# B&R Automation Studio project VerticalStacker
Automation Studio 4.10.2.37; technology packages: mappMotion 5.12.3, mappSafety 5.12.2

## Configuration Simulation

CPU X20cCP3586, AutomationRuntime B4.91, Build 4.1.2, Safety 0.0, Vc V4.72.3

### Task classes (Cpu.sw)
```
Cyclic#1:
  Program <- Program.prg
Libraries: SfDomain, standard, McBase, MpAxis, McAxis, MpBase, McAcpAx
```

### Hardware
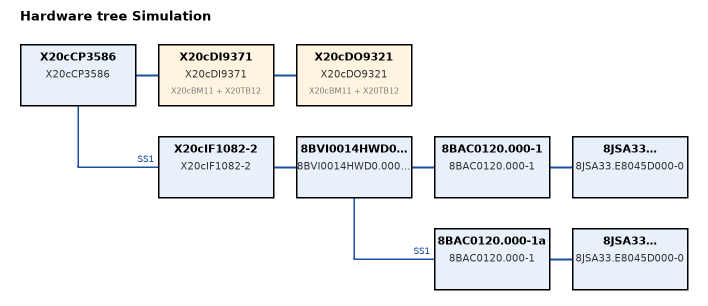
```
8BAC0120.000-1 : 8BAC0120.000-1 v2.2.0.0  [SS -> 8BVI0014HWD0.000-1.SS2]
  PlugInType = Encoder
  McAcoposTypeID = AcoposMultiPlugInConfig
8BAC0120.000-1a : 8BAC0120.000-1 v2.2.0.0  [SS -> 8BVI0014HWD0.000-1.SS1]
  PlugInType = Encoder
  McAcoposTypeID = AcoposMultiPlugInConfig
8BVI0014HWD0.000-1 : 8BVI0014HWD0.000-1 v2.3.0.1  [PLK1 -> X20cIF1082-2.IF1 (NodeNumber=1) [Cable Type=PowerlinkCable, Length=10, Version=1.0.0.3]; MT2 -> 8JSA33.E8045D000-0.MT]
  DriveConfiguration/Module:
    McAcoposTypeID = AcoposMultiDConfig
    ActivateACOPOSSimulationOnPLC = 1
    PowerSupply = ETA
  DriveConfiguration/Channel[1]/RealAxis:
    AxisReference = 
  DriveConfiguration/Channel[1]/RealAxis/MechanicalElements/Gearbox:
    InputIsReadOnly = 0
    Input = 1
    OutputIsReadOnly = 0
    Output = 1
  DriveConfiguration/Channel[1]/RealAxis/MechanicalElements/RotaryToLinearTransformation:
    ReferenceDistanceIsReadOnly = 0
    ReferenceDistance = 1
  DriveConfiguration/Channel[1]/RealAxis/Controller:
    ModeIsReadOnly = 0
    Mode = PositionController
  DriveConfiguration/Channel[1]/RealAxis/Controller/Mode/Position:
    ProportionalGain = 50.0
    IntegrationTime = 0.0
    PredictionTime = 0.0004
    TotalDelayTime = 0.0004
  DriveConfiguration/Channel[1]/RealAxis/Controller/Mode/Speed:
    ProportionalGainIsReadOnly = 0
    ProportionalGain = 2.0
    IntegrationTimeIsReadOnly = 0
    IntegrationTime = 0.0
    FilterTimeIsReadOnly = 0
    FilterTime = 0.0
  DriveConfiguration/Channel[1]/RealAxis/Controller/Mode/LoopFilters:
    LoopFilter1 = NotUsed
    LoopFilter2 = NotUsed
    LoopFilter3 = NotUsed
  DriveConfiguration/Channel[1]/RealAxis/Homing:
    Mode = Direct
  DriveConfiguration/Channel[1]/RealAxis/Homing/Mode:
    Position = 0.0
    ReferencePulse = NotUsed
  DriveConfiguration/Channel[1]/RealAxis/Homing:
    RestorePositionVariable = 
  DriveConfiguration/Channel[1]/RealAxis/StopReaction:
    Quickstop = DecelerationLimit
    DriveError = DecelerationLimit
  DriveConfiguration/Channel[1]/RealAxis/MovementErrorLimits:
    PositionError = 1.0
    VelocityErrorMonitoring = Automatic1
  DriveConfiguration/Channel[1]/RealAxis:
    JerkFilter = NotUsed
  DriveConfiguration/Channel[1]/RealAxis/DigitalInputs/HomingSwitch:
    Source = NotUsed
    Level = High
  DriveConfiguration/Channel[1]/RealAxis/DigitalInputs/PositiveLimitSwitch:
    Source = NotUsed
    Level = High
  DriveConfiguration/Channel[1]/RealAxis/DigitalInputs/NegativeLimitSwitch:
    Source = NotUsed
    Level = High
  DriveConfiguration/Channel[1]/RealAxis/DigitalInputs/Trigger1:
    Level = High
  DriveConfiguration/Channel[1]/RealAxis/DigitalInputs/Trigger2:
    Level = High
  DriveConfiguration/Channel[1]/RealAxis/DigitalInputs/Quickstop:
    Input = Trigger2
  DriveConfiguration/Channel[1]/RealAxis/Simulation:
    SimulationModeOnPLC = SetValueGeneration
    SimulationModeOnACOPOS = NotUsed
  DriveConfiguration/Channel[1]:
    VirtualAxis = Used
  DriveConfiguration/Channel[1]/VirtualAxis:
    AxisReference = gAxis_1
  DriveConfiguration/Channel[1]/VirtualAxis/Homing:
    Mode = Direct
  DriveConfiguration/Channel[1]/VirtualAxis/Homing/Mode:
    Position = 0.0
  DriveConfiguration/Channel[1]/VirtualAxis/Homing:
    RestorePositionVariable = 
  DriveConfiguration/Channel[1]/VirtualAxis:
    JerkFilter = NotUsed
  DriveConfiguration/Channel[2]/RealAxis:
    AxisReference = 
  DriveConfiguration/Channel[2]/RealAxis/MechanicalElements/Gearbox:
    InputIsReadOnly = 0
    Input = 1
    OutputIsReadOnly = 0
    Output = 1
  DriveConfiguration/Channel[2]/RealAxis/MechanicalElements/RotaryToLinearTransformation:
    ReferenceDistanceIsReadOnly = 0
    ReferenceDistance = 1
  DriveConfiguration/Channel[2]/RealAxis/Controller:
    ModeIsReadOnly = 0
    Mode = PositionController
  DriveConfiguration/Channel[2]/RealAxis/Controller/Mode/Position:
    ProportionalGain = 50.0
    IntegrationTime = 0.0
    PredictionTime = 0.0004
    TotalDelayTime = 0.0004
  DriveConfiguration/Channel[2]/RealAxis/Controller/Mode/Speed:
    ProportionalGainIsReadOnly = 0
    ProportionalGain = 2.0
    IntegrationTimeIsReadOnly = 0
    IntegrationTime = 0.0
    FilterTimeIsReadOnly = 0
    FilterTime = 0.0
  DriveConfiguration/Channel[2]/RealAxis/Controller/Mode/LoopFilters:
    LoopFilter1 = NotUsed
    LoopFilter2 = NotUsed
    LoopFilter3 = NotUsed
  DriveConfiguration/Channel[2]/RealAxis/Homing:
    Mode = Direct
  DriveConfiguration/Channel[2]/RealAxis/Homing/Mode:
    Position = 0.0
    ReferencePulse = NotUsed
  DriveConfiguration/Channel[2]/RealAxis/Homing:
    RestorePositionVariable = 
  DriveConfiguration/Channel[2]/RealAxis/StopReaction:
    Quickstop = DecelerationLimit
    DriveError = DecelerationLimit
  DriveConfiguration/Channel[2]/RealAxis/MovementErrorLimits:
    PositionError = 1.0
    VelocityErrorMonitoring = Automatic1
  DriveConfiguration/Channel[2]/RealAxis:
    JerkFilter = NotUsed
  DriveConfiguration/Channel[2]/RealAxis/DigitalInputs/HomingSwitch:
    Source = NotUsed
    Level = High
  DriveConfiguration/Channel[2]/RealAxis/DigitalInputs/PositiveLimitSwitch:
    Source = NotUsed
    Level = High
  DriveConfiguration/Channel[2]/RealAxis/DigitalInputs/NegativeLimitSwitch:
    Source = NotUsed
    Level = High
  DriveConfiguration/Channel[2]/RealAxis/DigitalInputs/Trigger1:
    Level = High
  DriveConfiguration/Channel[2]/RealAxis/DigitalInputs/Trigger2:
    Level = High
  DriveConfiguration/Channel[2]/RealAxis/DigitalInputs/Quickstop:
    Input = Trigger2
  DriveConfiguration/Channel[2]/RealAxis/Simulation:
    SimulationModeOnPLC = SetValueGeneration
    SimulationModeOnACOPOS = NotUsed
  DriveConfiguration/Channel[2]:
    VirtualAxis = Used
  DriveConfiguration/Channel[2]/VirtualAxis:
    AxisReference = gAxis_2
  DriveConfiguration/Channel[2]/VirtualAxis/Homing:
    Mode = Direct
  DriveConfiguration/Channel[2]/VirtualAxis/Homing/Mode:
    Position = 0.0
  DriveConfiguration/Channel[2]/VirtualAxis/Homing:
    RestorePositionVariable = 
  DriveConfiguration/Channel[2]/VirtualAxis:
    JerkFilter = NotUsed
8JSA33.E8045D000-0 : 8JSA33.E8045D000-0 v1.0.6.30  [EC -> 8BAC0120.000-1.EC; MT -> 8BVI0014HWD0.000-1.MT2]
8JSA33.E8045D000-0a : 8JSA33.E8045D000-0 v1.0.6.30  [EC -> 8BAC0120.000-1a.EC; MT -> 8BVI0014HWD0.000-1.MT1]
X20TB12 : X20TB12 v1.0.0.0
X20TB12a : X20TB12 v1.0.0.0
X20cBM11 : X20cBM11 v1.0.1.0  [X2X1 -> X20cCP3586.IF6]
X20cBM11a : X20cBM11 v1.0.1.0  [X2X1 -> X20cBM11.X2X2]
X20cCP3586 : X20cCP3586 v1.9.0.0
  Connector IF2:
    ActivateDevice = 1
  ConfigurationID = Project_VerticalStacker_Config1
  Simulation = 1
  FileDevice1
  FileDeviceName1 = USER
  FileDevicePath1 = USER_PATH
  ActivateOpcUa = 1
  OpcUaPort = 4842
  OpcUa_AuthenticationSecurityPolicy_EnableNone = 1
  OpcUa_AuthenticationSecurityPolicy_EnableBasic128Rsa15 = 1
  OpcUaInformationModels_PV_Version = 1
X20cDI9371 : X20cDI9371 v1.1.0.0  [SS1 -> X20TB12.SS; SL -> X20cBM11.SL1]
X20cDO9321 : X20cDO9321 v1.1.0.0  [SS1 -> X20TB12a.SS; SL -> X20cBM11a.SL1]
X20cIF1082-2 : X20cIF1082-2 v1.11.1.0  [SS -> X20cCP3586.SS1]
  Connector IF1:
    EplNatSubnet = 192.168.102.0
```

- Physical/Simulation/X20cCP3586/IoMap.iom: same as Physical/Simulation/X20cCP3586/Cpu.per
- Physical/Simulation/X20cCP3586/PvMap.vvm: same as Physical/Simulation/X20cCP3586/Cpu.per
### Config_1.axis - X20cCP3586/mappMotion/Config_1.axis
```
Element gAxis_1 (Type=axis)
  BaseTypeIsReadOnly = 0
  BaseType = LinearBounded
    MeasurementUnit = 5066068
    MeasurementResolutionIsReadOnly = 0
    MeasurementResolution = 0.01
    CountDirectionIsReadOnly = 0
    CountDirection = Standard
  MovementLimitsIsReadOnly = 0
  MovementLimits = Internal
    Position:
      LowerLimitMin = -1.79769313486231E308
      UpperLimitMax = 1.79769313486231E308
      LowerLimit = -1000.0
      UpperLimit = 1000.0
    VelocityIsReadOnly = 0
    Velocity:
      VelocityMax = 3.4E38
      Velocity = 10.0
    AccelerationIsReadOnly = 0
    Acceleration:
      AccelerationMax = 3.4E38
      Acceleration = 50.0
    DecelerationIsReadOnly = 0
    Deceleration:
      DecelerationMax = 3.4E38
      Deceleration = 50.0
  Alarms = None
Element gAxis_2 (Type=axis)
  BaseTypeIsReadOnly = 0
  BaseType = LinearBounded
    MeasurementUnit = 5066068
    MeasurementResolutionIsReadOnly = 0
    MeasurementResolution = 0.01
    CountDirectionIsReadOnly = 0
    CountDirection = Standard
  MovementLimitsIsReadOnly = 0
  MovementLimits = Internal
    Position:
      LowerLimitMin = -1.79769313486231E308
      UpperLimitMax = 1.79769313486231E308
      LowerLimit = -1000.0
      UpperLimit = 1000.0
    VelocityIsReadOnly = 0
    Velocity:
      VelocityMax = 3.4E38
      Velocity = 10.0
    AccelerationIsReadOnly = 0
    Acceleration:
      AccelerationMax = 3.4E38
      Acceleration = 50.0
    DecelerationIsReadOnly = 0
    Deceleration:
      DecelerationMax = 3.4E38
      Deceleration = 50.0
  Alarms = None
```

- Safety project (password-protected, skipped)

## Logical view

Binary libraries used (declarations not repeated): operator, runtime, astime, AsIecCon, SfDomain 5.12.2, standard, McBase 5.12.3, MpAxis 5.12.3, McAxis 5.12.3, MpBase 5.12.0, McAcpAx 5.12.3


### Program Logical/Program (IEC)

#### Main.st - Init, cyclic, exit code
```iecst
(*
Name					Date				Version				Note
Jamal Muhammad			10.10.2021			V2021.1				First version
*)

PROGRAM _INIT
	MpAxisBasic_0.Enable := TRUE;
	xHomingCmd := TRUE;

	AxisParameters.Velocity := 5.0;
	AxisParameters.Acceleration := 20.0;
	AxisParameters.Deceleration := 20.0;

	xPartLoadFirstCycle := TRUE;
	xPartUnloadFirstCycle := TRUE;
	// For simulation purpose
	FOR i:=1 TO 20 DO
		aBufferData[i].usiSeqNumber:= i;
		aBufferData[i].usiPartId := 100+i;
	END_FOR
	usiPartId := 120;
END_PROGRAM

PROGRAM _CYCLIC
	// Inputs
	lrServoPosition := MpAxisBasic_0.Position;

	stServoState.PowerON := MpAxisBasic_0.PowerOn;
	stServoState.Active := MpAxisBasic_0.Active;
	stServoState.MoveActive := MpAxisBasic_0.MoveActive;
	stServoState.Error := MpAxisBasic_0.Error;

	// Initialisation
	IF xInit = FALSE THEN
		ton_1(IN:=NOT ton_1.Q,PT:=T#3500MS);
		IF ton_1.Q THEN
			ton_1(IN:=FALSE,PT:=t#0MS);
			xInit := TRUE;
		END_IF
	END_IF

	//	Enabling/Disabling servo
	IF xServoError OR xEmergencyStopInactive_NC=FALSE OR xDriveStopInactive_NC=FALSE THEN
		xServoEnable:=FALSE;
	ELSE
		xServoEnable:=TRUE;
	END_IF

	// Enabling servo power automatically after initialisation & xServoEnable are ON
	IF xServoEnable AND xInit AND MpAxisBasic_0.PowerOn = FALSE THEN
		MpAxisBasic_0.Power := TRUE;
	END_IF

	// If xHomingCmd is ON then move servo to zero position
	IF MpAxisBasic_0.Position = 0 THEN
		xHomingCmd := FALSE;
	ELSIF MpAxisBasic_0.Position<>0 AND xHomingCmd = TRUE AND MpAxisBasic_0.PowerOn THEN
		AxisParameters.Position := 0.0;
		MpAxisBasic_0.MoveAbsolute := TRUE;
	END_IF;

	// Part unloading has priority-1, part unloading has priority-2
	IF xUnloadPartCmd THEN
		xLoadPartCmd := FALSE;
	END_IF

	//Check if buffer is full
	usiCounter := 0;
	FOR i:=1 TO usiPartBufferMax DO
		IF aBufferData[i].usiPartId <> 0 THEN
			usiCounter := usiCounter+1;
		END_IF
	END_FOR
	IF usiCounter = usiPartBufferMax THEN
		xBufferFull:=TRUE;
	ELSE
		xBufferFull:=FALSE;
	END_IF

	// State Machine > Unloading buffer
	IF xUnloadPartCmd AND xHomingCmd=FALSE AND MpAxisBasic_0.Enable THEN
		enumState_part_loading:=ST_LD_TO_ZERO_POS_1;
		xPartLoadFirstCycle:=TRUE;

		CASE enumState_part_unloading OF
			//*********************
			ST_UNLD_TO_ZERO_POS_1:
				IF xPartUnloadFirstCycle AND lrServoPosition<>0 THEN
					AxisParameters.Position := 0.0;
					AxisParameters.Velocity := 40.0;
					AxisParameters.Acceleration := 160.0;
					AxisParameters.Deceleration := 160.0;
					AxisUpdate;
					IF xAxisUpdateDone AND MpAxisBasic_0.MoveActive=FALSE THEN
						MpAxisBasic_0.MoveAbsolute := TRUE;
						enumState_part_unloading:=ST_UNLD_TO_ZERO_POS_2;
					END_IF
				ELSE
					enumState_part_unloading:=ST_UNLD_SET_AXIS_PARAMS_1;
				END_IF
			//*********************
			ST_UNLD_TO_ZERO_POS_2:
				IF lrServoPosition=0 THEN
					xPartUnloadFirstCycle := FALSE;
					MpAxisBasic_0.MoveAbsolute := FALSE;
					enumState_part_unloading:=ST_UNLD_SET_AXIS_PARAMS_1;
				END_IF
			//*********************
			ST_UNLD_SET_AXIS_PARAMS_1:
				IF lrServoPosition<690 AND MpAxisBasic_0.MoveActive=FALSE THEN
					AxisParameters.Position := 690.0;
					AxisParameters.Velocity := 10.0;
					AxisParameters.Acceleration := 40.0;
					AxisParameters.Deceleration := 40.0;
					AxisUpdate;
					IF xAxisUpdateDone THEN
						enumState_part_unloading:=ST_UNLD_IF_UNLOAD_CMD;
					END_IF
				END_IF
			//*********************
			ST_UNLD_IF_UNLOAD_CMD:
				IF xUnloadPartCmd THEN
					enumState_part_unloading:=ST_UNLD_FIND_UNLOADING_TARGET;
				END_IF
			//*********************
			ST_UNLD_FIND_UNLOADING_TARGET:
				FOR i:=1 TO usiPartBufferMax DO
					IF aBufferData[i].usiPartId <> 0 THEN
						FOR j:=1 TO usiPartBufferMax DO
							IF aBufferData[j].usiPartId<>0 AND i<>j AND aBufferData[i].usiPartId < aBufferData[j].usiPartId THEN
								usiTarget := i;
							ELSIF i=usiPartBufferMax THEN
								usiTarget := i;
							ELSE
								usiTarget := 0;
							END_IF
						END_FOR
						IF usiTarget<>0 THEN
							enumState_part_unloading:=ST_UNLD_SET_AXIS_PARAMS_2;
							EXIT;
						END_IF
					END_IF
				END_FOR
			//*********************
			ST_UNLD_SET_AXIS_PARAMS_2:
				AxisParameters.Position := usiTarget*34.5;
				AxisParameters.Velocity := 10.0;
				AxisParameters.Acceleration := 40.0;
				AxisParameters.Deceleration := 40.0;
				IF xAxisUpdateDone THEN
					enumState_part_unloading:=ST_UNLD_SERVO_MOVE_TO_TARGET;
				END_IF
			//*********************
			ST_UNLD_SERVO_MOVE_TO_TARGET:
				MpAxisBasic_0.MoveAbsolute := TRUE;

				IF AxisParameters.Position > lrServoPosition  THEN
					IF lrServoPosition > AxisParameters.Position-5 THEN
						MpAxisBasic_0.MoveAbsolute := FALSE;
						enumState_part_unloading:=ST_UNLD_SET_AXIS_PARAMS_3;
					END_IF;
				END_IF

				IF AxisParameters.Position < lrServoPosition  THEN
					IF lrServoPosition < AxisParameters.Position+5 THEN
						MpAxisBasic_0.MoveAbsolute := FALSE;
						enumState_part_unloading:=ST_UNLD_SET_AXIS_PARAMS_3;
					END_IF;
				END_IF
			//*********************
			ST_UNLD_SET_AXIS_PARAMS_3:
				IF MpAxisBasic_0.MoveActive = FALSE THEN
					AxisParameters.Velocity := 1.0;
					AxisParameters.Acceleration := 4.0;
					AxisParameters.Deceleration := 4.0;
					AxisUpdate;
					IF xAxisUpdateDone THEN
						enumState_part_unloading:=ST_UNLD_SERVO_MOVE_SLOW;
					END_IF
				END_IF
			//*********************
			ST_UNLD_SERVO_MOVE_SLOW:
				MpAxisBasic_0.MoveAbsolute := TRUE;
				IF lrServoPosition=usiTarget*34.5 THEN
					MpAxisBasic_0.MoveAbsolute := FALSE;
					enumState_part_unloading:=ST_UNLD_UPDATE_BUFFER_INFO;
				END_IF
			//*********************
			ST_UNLD_UPDATE_BUFFER_INFO:
				aBufferData[usiTarget].usiPartId:=0;
				IF xPartUnloaded THEN
					enumState_part_unloading:=ST_UNLD_DELAY;
				END_IF
			//*********************
			ST_UNLD_DELAY:
				ton_1(IN:=NOT ton_1.Q,PT:=T#750MS);
				IF ton_1.Q AND MpAxisBasic_0.MoveActive=FALSE THEN
					enumState_part_unloading:=ST_UNLD_IF_UNLOAD_CMD;
				END_IF
		END_CASE
	END_IF

	// Loading buffer
	IF 	xLoadPartCmd
		AND MpAxisBasic_0.Enable
		AND xHomingCmd=FALSE
		AND xBufferFull=FALSE THEN
		enumState_part_unloading:=ST_UNLD_TO_ZERO_POS_1;
			xPartUnloadFirstCycle:=TRUE;

		CASE enumState_part_loading OF
			//*********************
			ST_LD_TO_ZERO_POS_1:
				IF xPartLoadFirstCycle AND lrServoPosition<>0 THEN
					AxisParameters.Position := 0.0;
					AxisParameters.Velocity := 40.0;
					AxisParameters.Acceleration := 160.0;
					AxisParameters.Deceleration := 160.0;
					AxisUpdate;
					IF xAxisUpdateDone THEN
						MpAxisBasic_0.MoveAbsolute := TRUE;
						enumState_part_loading:=ST_LD_TO_ZERO_POS_2;
					END_IF
				ELSE
					enumState_part_loading:=ST_LD_SET_AXIS_PARAMS_1;
				END_IF
			//*********************
			ST_LD_TO_ZERO_POS_2:
				IF lrServoPosition=0 THEN
					xPartLoadFirstCycle := FALSE;
					MpAxisBasic_0.MoveAbsolute := FALSE;
					enumState_part_loading:=ST_LD_SET_AXIS_PARAMS_1;
				END_IF
			//*********************
			ST_LD_SET_AXIS_PARAMS_1:
				IF lrServoPosition<690 AND MpAxisBasic_0.MoveActive = FALSE THEN
					AxisParameters.Position := 690.0;
					AxisParameters.Velocity := 10.0;
					AxisParameters.Acceleration := 40.0;
					AxisParameters.Deceleration := 40.0;
					AxisUpdate;
					IF xAxisUpdateDone THEN
						enumState_part_loading:=ST_LD_FIND_LOADING_TARGET;
					END_IF
				END_IF
			//*********************
			ST_LD_FIND_LOADING_TARGET:
				FOR i:=1 TO 20 DO
					IF aBufferData[i].usiPartId = 0 THEN
						usiTarget := i;
						enumState_part_loading:=ST_LD_SERVO_MOVE_FAST;
						EXIT;
					END_IF
				END_FOR
			//*********************
			ST_LD_SERVO_MOVE_FAST:
				MpAxisBasic_0.MoveAbsolute := TRUE;

				IF lrServoPosition>((usiTarget*34.5)-4)THEN
					MpAxisBasic_0.MoveAbsolute := FALSE;
					enumState_part_loading:=ST_LD_SET_AXIS_PARAMS_2;
				END_IF
			//*********************
			ST_LD_SET_AXIS_PARAMS_2:
				IF MpAxisBasic_0.MoveActive = FALSE THEN
					AxisParameters.Velocity := 1.0;
					AxisParameters.Acceleration := 4.0;
					AxisParameters.Deceleration := 4.0;
					AxisUpdate;
					IF xAxisUpdateDone THEN
						enumState_part_loading:=ST_LD_SERVO_MOVE_SLOW;
					END_IF
				END_IF
			//*********************
			ST_LD_SERVO_MOVE_SLOW:
				MpAxisBasic_0.MoveAbsolute := TRUE;

				IF ((lrServoPosition=usiTarget*34.5) OR (lrServoPosition>(usiTarget*34.5))) THEN
					MpAxisBasic_0.MoveAbsolute := FALSE;
					enumState_part_loading:=ST_LD_UPDATE_BUFFER_INFO_1;
				END_IF
			//*********************
			ST_LD_UPDATE_BUFFER_INFO_1:
				IF aBufferData[usiTarget].usiPartId = 0 THEN
					enumState_part_loading:=ST_LD_UPDATE_BUFFER_INFO_2;
				END_IF
			//*********************
			ST_LD_UPDATE_BUFFER_INFO_2:
				IF xPartLoaded THEN
					usiPartId := usiPartId+1;
					aBufferData[usiTarget].usiPartId:=usiPartId;
					enumState_part_loading:=ST_LD_DELAY;
				END_IF
			//*********************
			ST_LD_DELAY:
				ton_1(IN:=NOT ton_1.Q,PT:=T#750MS);
				IF ton_1.Q AND MpAxisBasic_0.MoveActive=FALSE THEN
					ton_1(IN:=FALSE,PT:=T#0MS);
					enumState_part_loading:=ST_LD_SET_AXIS_PARAMS_1;
				END_IF
		END_CASE
	END_IF

	// Servo axis movement command
	MpAxisBasic_0.MpLink     := ADR(gAxis_1);
	MpAxisBasic_0.Parameters := ADR(AxisParameters);
	MpAxisBasic_0();

	// Outputs
	IF xUnloadPartCmd=FALSE AND xLoadPartCmd=FALSE AND xHomingCmd = FALSE THEN
		MpAxisBasic_0.MoveAbsolute := FALSE;
	END_IF

END_PROGRAM

PROGRAM _EXIT
	;
END_PROGRAM
```

#### Types.typ - Local data types
```iecst
TYPE
	STATE_PART_LOADING :
		(
		ST_LD_TO_ZERO_POS_1,
		ST_LD_TO_ZERO_POS_2,
		ST_LD_SET_AXIS_PARAMS_1,
		ST_LD_FIND_LOADING_TARGET,
		ST_LD_SERVO_MOVE_FAST,
		ST_LD_SET_AXIS_PARAMS_2,
		ST_LD_SERVO_MOVE_SLOW,
		ST_LD_UPDATE_BUFFER_INFO_1,
		ST_LD_UPDATE_BUFFER_INFO_2,
		ST_LD_DELAY,
		ST_LD_ERROR
		);
	STATE_PART_UNLOADING :
		(
		ST_UNLD_TO_ZERO_POS_1,
		ST_UNLD_TO_ZERO_POS_2,
		ST_UNLD_SET_AXIS_PARAMS_1,
		ST_UNLD_IF_UNLOAD_CMD,
		ST_UNLD_FIND_UNLOADING_TARGET,
		ST_UNLD_SET_AXIS_PARAMS_2,
		ST_UNLD_SERVO_MOVE_TO_TARGET,
		ST_UNLD_SET_AXIS_PARAMS_3,
		ST_UNLD_SERVO_MOVE_SLOW,
		ST_UNLD_UPDATE_BUFFER_INFO,
		ST_UNLD_DELAY,
		ST_UNLD_ERROR
		);
	HolderData : 	STRUCT
		usiSeqNumber : USINT;
		usiPartId : USINT;
	END_STRUCT;
	ServoState : 	STRUCT
		Active : BOOL;
		MoveActive : BOOL;
		PowerON : BOOL;
		Error : BOOL;
	END_STRUCT;
END_TYPE
```

#### Variables.var - Local variables
```iecst
VAR
	(*STRING*)
	strMachineID : STRING[80] := 'VB_L2_M12';
	(*BOOL*)
	xLoadPartCmd : BOOL;
	xUnloadPartCmd : BOOL;
	xPartLoaded : BOOL;
	xPartUnloaded : BOOL;
	xPartLoadFirstCycle : BOOL;
	xPartUnloadFirstCycle : BOOL;
	xAxisUpdateDone : BOOL;
	xInit : BOOL;
	xHomingCmd : BOOL;
	xServoEnable : BOOL;
	xServoError : BOOL;
	xBufferFull : BOOL;
	xEmergencyStopInactive_NC : BOOL := TRUE; (*Normally Closed(NC)*)
	xDriveStopInactive_NC : BOOL := TRUE; (*Normally Closed(NC)*)
	(*INTEGER*)
	i : USINT;
	j : USINT;
	usiCounter : USINT;
	usiTarget : USINT;
	usiPartId : USINT;
	(*REAL*)
	lrServoPosition : LREAL;
	(*TIMER*)
	ton_1 : {REDUND_UNREPLICABLE} TON;
	(*ARRAY*)
	aServoMoveMode : ARRAY[1..2] OF BOOL; (*ARRAY[1]=Manual mode free, ARRAY[2]=Manual mode step,ARRAY[3]=Automatic mode *)
	aBufferData : ARRAY[1..usiPartBufferMax] OF HolderData;
	(*ENUM*)
	enumState_part_loading : STATE_PART_LOADING;
	enumState_part_unloading : STATE_PART_UNLOADING;
	(*STRUCT*)
	stServoState : ServoState;
	(*INSTANCES*)
	MpAxisBasic_0 : MpAxisBasic;
	AxisParameters : MpAxisBasicParType;
	(*FUNCTION BLOCK*)

END_VAR

VAR CONSTANT
	usiPartBufferMax : USINT := 20;
END_VAR
```

#### AxisUpdate.st
```iecst
ACTION AxisUpdate:
	xAxisUpdateDone:=FALSE;

END_ACTION
```
